# EPICS substitutions: gp08_ioc01/gp08_ioc01App/Db/healthMonitor.substitutions
file elinp-iocmon.db
{
pattern { P                 }
        { GEN-CS-GP08:IOC01 }
}
file elinp-sysmon.db
{
pattern { P                 , NETIF }
        { GEN-CS-GP08:IOC01 , eth0  }
}
